Yaskawa INFORM job: WORKPIECE3.JBI

/JOB
//NAME WORKPIECE3
///FOLDERNAME INNE
//POS
///NPOS 9,9,0,0,0,0
///TOOL 0
///POSTYPE PULSE
///PULSE
C00000=34846,18001,86937,93778,55325,-59342
C00001=34431,-29522,5152,76593,58706,-45262
C00002=35202,-53816,-63523,62971,69519,-31037
C00003=115817,3588,31827,-1404,92004,-1585
C00004=147487,12091,39236,7520,90657,8603
C00005=193736,9628,36810,-20992,59161,-53276
C00006=109997,-133094,-95290,112234,-61835,-40831
C00007=110238,-102285,-50863,105980,-58681,-34982
C00008=110499,-37520,45015,89461,-56291,-21018
BC00000=3493,452410,917391
BC00001=3492,452410,1075223
BC00002=3492,452410,1075223
BC00003=298495,436540,859658
BC00004=298495,436540,859658
BC00005=298495,436540,859658
BC00006=4213,75267,1058272
BC00007=4213,75267,1058272
BC00008=4213,75267,1058272
//INST
///DATE 2023/10/04 15:16
///ATTR SC,RW
///GROUP1 RB1,BS1
NOP
'LEFT_SIDE
MOVJ C00000 BC00000 VJ=0.78 PL=0  //POINT1
MOVJ C00001 BC00001 VJ=0.78 PL=0  //POINT2
MOVJ C00002 BC00002 VJ=0.78 PL=0  //POINT3
'LEFT_2
MOVJ C00003 BC00003 VJ=0.78 PL=0  //POINT1
MOVJ C00004 BC00004 VJ=0.78 PL=0  //POINT2
MOVJ C00005 BC00005 VJ=0.78 PL=0  //POINT3
'BACK_SIDE
MOVJ C00006 BC00006 VJ=0.78 PL=0  //POINT1
MOVJ C00007 BC00007 VJ=0.78 PL=0  //POINT2
MOVJ C00008 BC00008 VJ=0.78 PL=0  //POINT3
END
